// TwinCAT 3 PLC project TcUnitVerifier
// Title: TcUnit verifier
// Company: www.tcunit.org
// Author: Jakob Sagatowski and other contributors, see CONTRIBUTORS file on www.github.com/tcunit/TcUnit-Verifier
// ProjectVersion: 0.5.0.0
// Description: This project is can be used to verify the different functions of TcUnit. It has various test suites to test different functions in TcUnit. By making sure to comment out everything except the test suite that is interesting it is possible to test only the specific function of TcUnit that is interesting.
// ProgramVersion: 3.1.4022.4
// libraries:
//   Tc2_Standard, * (Beckhoff Automation GmbH)
//   Tc2_System, * (Beckhoff Automation GmbH)
//   Tc3_Module, * (Beckhoff Automation GmbH)
//   TcUnit, * (www.tcunit.org)
// project tree:
//   / FB_AdjustAssertFailureMessageToMax252CharLength_Test.TcPOU (not stored), PlcTask.TcTTO
//   Test/ FB_AnyToUnionValue_Test.TcPOU, FB_ArrayPrimitiveTypes_Test.TcPOU, FB_AssertEveryFailedTestTwice.TcPOU, FB_AssertEveryFailedTestTwice_ArrayVersion.TcPOU, FB_CreateFourTestsWithSameName.TcPOU, FB_CreateDisabledTest.TcPOU, FB_MultipleAssertWithSameParametersInDifferentCyclesAndInSameTest.TcPOU, FB_MultipleAssertWithSameParametersInSameCycleWithSameTest.TcPOU, FB_MultipleAssertWithSameParametersInDifferentCyclesButWithDifferentTests.TcPOU, FB_PrimitiveTypes_Test.TcPOU, FB_AssertTrueFalse_Test.TcPOU, FB_AnyPrimitiveTypes_Test.TcPOU, PRG_TEST.TcPOU
// real-time tasks:
//   TASK PlcTask: cycle T#10ms, priority 20, ADS port 350

CONFIGURATION TcUnitVerifier
    RESOURCE PLC ON TwinCAT3
        TASK PlcTask(INTERVAL := T#10ms, PRIORITY := 20);
        PROGRAM PRG_TEST WITH PlcTask : PRG_TEST;
    END_RESOURCE
END_CONFIGURATION

// ---- Test/PRG_TEST.TcPOU
PROGRAM PRG_TEST
VAR
    PrimitiveTypesTest : FB_PrimitiveTypes_Test;
    AssertTrueFalse_Test : FB_AssertTrueFalse_Test;
    AssertEveryFailedTestTwice : FB_AssertEveryFailedTestTwice;
    CreateFourTestsWithSameName : FB_CreateFourTestsWithSameName;
    ArrayPrimitiveTypes_Test : FB_ArrayPrimitiveTypes_Test;
    CreateDisabledTest : FB_CreateDisabledTest;
    AnyPrimitiveTypes_Test : FB_AnyPrimitiveTypes_Test;
    AssertEveryFailedTestTwice_ArrayVersion : FB_AssertEveryFailedTestTwice_ArrayVersion;
    AnyToUnionValue_Test : FB_AnyToUnionValue_Test;
    MultipleAssertWithSameParametersInSameCycleWithSameTest : FB_MultipleAssertWithSameParametersInSameCycleWithSameTest;
    MultipleAssertWithSameParametersInDifferentCyclesButWithDifferentTests : FB_MultipleAssertWithSameParametersInDifferentCyclesButWithDifferentTests;
    MultipleAssertWithSameParametersInDifferentCyclesAndInSameTest : FB_MultipleAssertWithSameParametersInDifferentCyclesAndInSameTest;
END_VAR

TcUnit.RUN();

END_PROGRAM

// ---- Test/FB_PrimitiveTypes_Test.TcPOU
(*
    This testsuite tests the different assert-functions for all the different data types in TwinCAT.
    For every data type at least two different tests have been defined:
        1. One test that succeeds (Expected and actual are equal)
        2. One test that fails (Expected and actual are false).
*)
{attribute 'call_after_init'}
FUNCTION_BLOCK FB_PrimitiveTypes_Test EXTENDS TcUnit.FB_TestSuite

Test_ANY_Equals();
Test_ANY_Differ_DataType();
Test_BYTE_Equals();
Test_BYTE_Differ();
Test_BOOL_Equals();
Test_BOOL_Differ();
Test_DATE_Equals();
Test_DATE_Differ();
Test_DATE_AND_TIME_Equals();
Test_DATE_AND_TIME_Differ();
Test_DINT_Equals();
Test_DINT_Differ();
Test_DWORD_Equals();
Test_DWORD_Differ();
Test_INT_Equals();
Test_INT_Differ();
Test_LINT_Equals();
Test_LINT_Differ();
Test_LREAL_Equals();
Test_LREAL_Differ();
Test_LTIME_Equals();
Test_LTIME_Differ();
Test_LWORD_Equals();
Test_LWORD_Differ();
Test_REAL_Equals();
Test_REAL_Differ();
Test_SINT_Equals();
Test_SINT_Differ();
Test_STRING_Equals();
Test_STRING_Differ();
Test_TIME_Equals();
Test_TIME_Differ();
Test_TIME_OF_DAY_Equals();
Test_TIME_OF_DAY_Differ();
Test_UDINT_Equals();
Test_UDINT_Differ();
Test_UINT_Equals();
Test_UINT_Differ();
Test_ULINT_Equals();
Test_ULINT_Differ();
Test_USINT_Equals();
Test_USINT_Differ();
Test_WORD_Equals();
Test_WORD_Differ();

METHOD PRIVATE Test_ANY_Differ_DataType
VAR
    a : INT := 5;
    b : UINT := 5;
END_VAR
TEST('Test_ANY_Differ_DataType');

AssertEquals(Expected := a,
             Actual := b,
             Message := 'Values differ');

TEST_FINISHED();
END_METHOD

METHOD PRIVATE Test_ANY_Equals
VAR
    a : INT := 5;
    b : INT := 5;
END_VAR
TEST('Test_ANY_Equals');

AssertEquals(Expected := a,
             Actual := b,
             Message := 'Values differ');

TEST_FINISHED();
END_METHOD

METHOD PRIVATE Test_BOOL_Differ
VAR
    a : BOOL := TRUE;
    b : BOOL := FALSE;
END_VAR
TEST('Test_BOOL_Differ');

AssertEquals_BOOL(Expected := a,
                  Actual := b,
                  Message := 'Values differ');

TEST_FINISHED();
END_METHOD

METHOD PRIVATE Test_BOOL_Equals
VAR
    a : BOOL := TRUE;
    b : BOOL := TRUE;
END_VAR
TEST('Test_BOOL_Equals');

AssertEquals_BOOL(Expected := a,
                  Actual := b,
                  Message := 'Values differ');

TEST_FINISHED();
END_METHOD

METHOD PRIVATE Test_BYTE_Differ
VAR
    a : BYTE := 16#AB;
    b : BYTE := 16#CD;
END_VAR
TEST('Test_BYTE_Differ');

AssertEquals_BYTE(Expected := a,
                  Actual := b,
                  Message := 'Values differ');

TEST_FINISHED();
END_METHOD

METHOD PRIVATE Test_BYTE_Equals
VAR
    a : BYTE := 16#CD;
    b : BYTE := 16#CD;
END_VAR
TEST('Test_BYTE_Equals');

AssertEquals_BYTE(Expected := a,
                  Actual := b,
                  Message := 'Values differ');
TEST_FINISHED();
END_METHOD

METHOD PRIVATE Test_DATE_AND_TIME_Differ
VAR
    a : DATE_AND_TIME := DATE_AND_TIME#1996-05-06-15:36:30;
    b : DATE_AND_TIME := DATE_AND_TIME#1972-03-29-00:00:00;
END_VAR
TEST('Test_DATE_AND_TIME_Differ');

AssertEquals_DATE_AND_TIME(Expected := a,
                           Actual := b,
                           Message := 'Values differ');

TEST_FINISHED();
END_METHOD

METHOD PRIVATE Test_DATE_AND_TIME_Equals
VAR
    a : DATE_AND_TIME := DATE_AND_TIME#2019-01-20-13:54:30;
    b : DATE_AND_TIME := DATE_AND_TIME#2019-01-20-13:54:30;
END_VAR
TEST('Test_DATE_AND_TIME_Equals');

AssertEquals_DATE_AND_TIME(Expected := a,
                           Actual := b,
                           Message := 'Values differ');

TEST_FINISHED();
END_METHOD

METHOD PRIVATE Test_DATE_Differ
VAR
    a : DATE := DATE#1996-05-06;
    b : DATE := DATE#2019-01-20;
END_VAR
TEST('Test_DATE_Differ');

AssertEquals_DATE(Expected := a,
                  Actual := b,
                  Message := 'Values differ');

TEST_FINISHED();
END_METHOD

METHOD PRIVATE Test_DATE_Equals
VAR
    a : DATE := DATE#1996-05-06;
    b : DATE := DATE#1996-05-06;
END_VAR
TEST('Test_DATE_Equals');

AssertEquals_DATE(Expected := a,
                  Actual := b,
                  Message := 'Values differ');

TEST_FINISHED();
END_METHOD

METHOD PRIVATE Test_DINT_Differ
VAR
    a : DINT := -55555;
    b : DINT := 70000;
END_VAR
TEST('Test_DINT_Differ');

AssertEquals_DINT(Expected := a,
                  Actual := b,
                  Message := 'Values differ');

TEST_FINISHED();
END_METHOD

METHOD PRIVATE Test_DINT_Equals
VAR
    a : DINT := -80000;
    b : DINT := -80000;
END_VAR
TEST('Test_DINT_Equals');

AssertEquals_DINT(Expected := a,
                  Actual := b,
                  Message := 'Values differ');

TEST_FINISHED();
END_METHOD

METHOD PRIVATE Test_DWORD_Differ
VAR
    a : DWORD := 16#12345678;
    b : DWORD := 16#90ABCDEF;
END_VAR
TEST('Test_DWORD_Differ');

AssertEquals_DWORD(Expected := a,
                   Actual := b,
                   Message := 'Values differ');

TEST_FINISHED();
END_METHOD

METHOD PRIVATE Test_DWORD_Equals
VAR
    a : DWORD := 16#7890ABCD;
    b : DWORD := 16#7890ABCD;
END_VAR
TEST('Test_DWORD_Equals');

AssertEquals_DWORD(Expected := a,
                   Actual := b,
                   Message := 'Values differ');

TEST_FINISHED();
END_METHOD

METHOD PRIVATE Test_INT_Differ
VAR
    a : INT := -32000;
    b : INT := 15423;
END_VAR
TEST('Test_INT_Differ');

AssertEquals_INT(Expected := a,
                 Actual := b,
                 Message := 'Values differ');

TEST_FINISHED();
END_METHOD

METHOD PRIVATE Test_INT_Equals
VAR
    a : INT := -12345;
    b : INT := -12345;
END_VAR
TEST('Test_INT_Equals');

AssertEquals_INT(Expected := a,
                 Actual := b,
                 Message := 'Values differ');

TEST_FINISHED();
END_METHOD

METHOD PRIVATE Test_LINT_Differ
VAR
    a : LINT := -451416345;
    b : LINT := 589532453;
END_VAR
TEST('Test_LINT_Differ');

AssertEquals_LINT(Expected := a,
                  Actual := b,
                  Message := 'Values differ');

TEST_FINISHED();
END_METHOD

METHOD PRIVATE Test_LINT_Equals
VAR
    a : LINT := -123456789;
    b : LINT := -123456789;
END_VAR
TEST('Test_LINT_Equals');

AssertEquals_LINT(Expected := a,
                  Actual := b,
                  Message := 'Values differ');

TEST_FINISHED();
END_METHOD

METHOD PRIVATE Test_LREAL_Differ
VAR
    a : LREAL := 1234567.89;
    b : LREAL := 1234567.76;
END_VAR
TEST('Test_LREAL_Differ');

AssertEquals_LREAL(Expected := a,
                   Actual := b,
                   Delta := 0.1,
                   Message := 'Values differ');

TEST_FINISHED();
END_METHOD

METHOD PRIVATE Test_LREAL_Equals
VAR
    a : LREAL := 1234567.89;
    b : LREAL := 1234567.76;
END_VAR
TEST('Test_LREAL_Equals');

AssertEquals_LREAL(Expected := a,
                   Actual := b,
                   Delta := 0.2,
                   Message := 'Values differ');

TEST_FINISHED();
END_METHOD

METHOD PRIVATE Test_LTIME_Differ
VAR
    a : LTIME := LTIME#213503D23H34M33S709MS551US615NS;
    b : LTIME := LTIME#1000D15H23M12S34MS2US44NS;
END_VAR
TEST('Test_LTIME_Differ');

AssertEquals_LTIME(Expected := a,
                   Actual := b,
                   Message := 'Values differ');

TEST_FINISHED();
END_METHOD

METHOD PRIVATE Test_LTIME_Equals
VAR
    a : LTIME := LTIME#213503D23H34M33S709MS551US615NS;
    b : LTIME := LTIME#213503D23H34M33S709MS551US615NS;
END_VAR
TEST('Test_LTIME_Equals');

AssertEquals_LTIME(Expected := a,
                   Actual := b,
                   Message := 'Values differ');

TEST_FINISHED();
END_METHOD

METHOD PRIVATE Test_LWORD_Differ
VAR
    a : LWORD := 16#0123656789ABCBEC;
    b : LWORD := 16#0123256789ABCAEE;
END_VAR
TEST('Test_LWORD_Differ');

AssertEquals_LWORD(Expected := a,
                   Actual := b,
                   Message := 'Values differ');

TEST_FINISHED();
END_METHOD

METHOD PRIVATE Test_LWORD_Equals
VAR
    a : LWORD := 16#0123456789ABCDEF;
    b : LWORD := 16#0123456789ABCDEF;
END_VAR
TEST('Test_LWORD_Equals');

AssertEquals_LWORD(Expected := a,
                   Actual := b,
                   Message := 'Values differ');

TEST_FINISHED();
END_METHOD

METHOD PRIVATE Test_REAL_Differ
VAR
    a : REAL := 1234.5;
    b : REAL := 1234.4;
END_VAR
TEST('Test_REAL_Differ');

AssertEquals_REAL(Expected := a,
                  Actual := b,
                  Delta := 0.05,
                  Message := 'Values differ');

TEST_FINISHED();
END_METHOD

METHOD PRIVATE Test_REAL_Equals
VAR
    a : REAL := 1234.5;
    b : REAL := 1234.4;
END_VAR
TEST('Test_REAL_Equals');

AssertEquals_REAL(Expected := a,
                  Actual := b,
                  Delta := 0.1,
                  Message := 'Values differ');

TEST_FINISHED();
END_METHOD

METHOD PRIVATE Test_SINT_Differ
VAR
    a : SINT := 127;
    b : SINT := -30;
END_VAR
TEST('Test_SINT_Differ');

AssertEquals_SINT(Expected := a,
                  Actual := b,
                  Message := 'Values differ');

TEST_FINISHED();
END_METHOD

METHOD PRIVATE Test_SINT_Equals
VAR
    a : SINT := -128;
    b : SINT := -128;
END_VAR
TEST('Test_SINT_Equals');

AssertEquals_SINT(Expected := a,
                  Actual := b,
                  Message := 'Values differ');

TEST_FINISHED();
END_METHOD

METHOD PRIVATE Test_STRING_Differ
VAR
    a : STRING := 'This is a string';
    b : STRING := 'This is another string';
END_VAR
TEST('Test_STRING_Differ');

AssertEquals_STRING(Expected := a,
                    Actual := b,
                    Message := 'Values differ');

TEST_FINISHED();
END_METHOD

METHOD PRIVATE Test_STRING_Equals
VAR
    a : STRING := 'Hello there';
    b : STRING := 'Hello there';
END_VAR
TEST('Test_STRING_Equals');

AssertEquals_STRING(Expected := a,
                    Actual := b,
                    Message := 'Values differ');

TEST_FINISHED();
END_METHOD

METHOD PRIVATE Test_TIME_Differ
VAR
    a : TIME := T#12H34M15S10MS;
    b : TIME := T#11H34M13S244MS;
END_VAR
TEST('Test_TIME_Differ');

AssertEquals_TIME(Expected := a,
                  Actual := b,
                  Message := 'Values differ');

TEST_FINISHED();
END_METHOD

METHOD PRIVATE Test_TIME_Equals
VAR
    a : TIME := T#11H34M13S244MS;
    b : TIME := T#11H34M13S244MS;
END_VAR
TEST('Test_TIME_Equals');

AssertEquals_TIME(Expected := a,
                  Actual := b,
                  Message := 'Values differ');

TEST_FINISHED();
END_METHOD

METHOD PRIVATE Test_TIME_OF_DAY_Differ
VAR
    a : TIME_OF_DAY := TIME_OF_DAY#15:36:30.123;
    b : TIME_OF_DAY := TIME_OF_DAY#06:21:11.492;
END_VAR
TEST('Test_TIME_OF_DAY_Differ');

AssertEquals_TIME_OF_DAY(Expected := a,
                         Actual := b,
                         Message := 'Values differ');

TEST_FINISHED();
END_METHOD

METHOD PRIVATE Test_TIME_OF_DAY_Equals
VAR
    a : TIME_OF_DAY := TIME_OF_DAY#06:21:11.492;
    b : TIME_OF_DAY := TIME_OF_DAY#06:21:11.492;
END_VAR
TEST('Test_TIME_OF_DAY_Equals');

AssertEquals_TIME_OF_DAY(Expected := a,
                         Actual := b,
                         Message := 'Values differ');

TEST_FINISHED();
END_METHOD

METHOD PRIVATE Test_UDINT_Differ
VAR
    a : UDINT := 34124214;
    b : UDINT := 52343244;
END_VAR
TEST('Test_UDINT_Differ');

AssertEquals_UDINT(Expected := a,
                   Actual := b,
                   Message := 'Values differ');

TEST_FINISHED();
END_METHOD

METHOD PRIVATE Test_UDINT_Equals
VAR
    a : UDINT := 21845123;
    b : UDINT := 21845123;
END_VAR
TEST('Test_UDINT_Equals');

AssertEquals_UDINT(Expected := a,
                   Actual := b,
                   Message := 'Values differ');

TEST_FINISHED();
END_METHOD

METHOD PRIVATE Test_UINT_Differ
VAR
    a : UINT := 64322;
    b : UINT := 32312;
END_VAR
TEST('Test_UINT_Differ');

AssertEquals_UINT(Expected := a,
                  Actual := b,
                  Message := 'Values differ');

TEST_FINISHED();
END_METHOD

METHOD PRIVATE Test_UINT_Equals
VAR
    a : UINT := 65535;
    b : UINT := 65535;
END_VAR
TEST('Test_UINT_Equals');

AssertEquals_UINT(Expected := a,
                  Actual := b,
                  Message := 'Values differ');

TEST_FINISHED();
END_METHOD

METHOD PRIVATE Test_ULINT_Differ
VAR
    a : ULINT := 10000;
    b : ULINT := 53685437234;
END_VAR
TEST('Test_ULINT_Differ');

AssertEquals_ULINT(Expected := a,
                   Actual := b,
                   Message := 'Values differ');

TEST_FINISHED();
END_METHOD

METHOD PRIVATE Test_ULINT_Equals
VAR
    a : ULINT := 45683838383;
    b : ULINT := 45683838383;
END_VAR
TEST('Test_ULINT_Equals');

AssertEquals_ULINT(Expected := a,
                   Actual := b,
                   Message := 'Values differ');

TEST_FINISHED();
END_METHOD

METHOD PRIVATE Test_USINT_Differ
VAR
    a : USINT := 3;
    b : USINT := 7;
END_VAR
TEST('Test_USINT_Differ');

AssertEquals_USINT(Expected := a,
                   Actual := b,
                   Message := 'Values differ');

TEST_FINISHED();
END_METHOD

METHOD PRIVATE Test_USINT_Equals
VAR
    a : USINT := 5;
    b : USINT := 5;
END_VAR
TEST('Test_USINT_Equals');

AssertEquals_USINT(Expected := a,
                   Actual := b,
                   Message := 'Values differ');

TEST_FINISHED();
END_METHOD

METHOD PRIVATE Test_WORD_Differ
VAR
    a : WORD := 16#EF01;
    b : WORD := 16#2345;
END_VAR
TEST('Test_WORD_Differ');

AssertEquals_WORD(Expected := a,
                  Actual := b,
                  Message := 'Values differ');

TEST_FINISHED();
END_METHOD

METHOD PRIVATE Test_WORD_Equals
VAR
    a : WORD := 16#ABCD;
    b : WORD := 16#ABCD;
END_VAR
TEST('Test_WORD_Equals');

AssertEquals_WORD(Expected := a,
                  Actual := b,
                  Message := 'Values differ');

TEST_FINISHED();
END_METHOD

END_FUNCTION_BLOCK

// ---- Test/FB_AssertTrueFalse_Test.TcPOU
(* 
    This testsuite verifies that the Assert_True and Assert_False methods do what they are supposed to. It does so
    by making sure that every assert-method (assert_true & assert_false) does both one failing and one successful
    assert.
*)
{attribute 'call_after_init'}
FUNCTION_BLOCK FB_AssertTrueFalse_Test EXTENDS TcUnit.FB_TestSuite IMPLEMENTS TcUnit.I_RunnableTestSuite
VAR
    Assert : TcUnit.FB_Assert;
END_VAR

METHOD PRIVATE AssertThatINTsAreEqual
VAR
    a : INT := -33;
    b : INT := -44;
END_VAR
TEST('AssertThatINTsAreEqual');

Assert.AssertFalse(Condition := (a <> b),
                   Message := 'INTs are equal');
END_METHOD

METHOD PRIVATE AssertThatINTsAreNotEqual
VAR
    a : INT := -33;
    b : INT := -44;
END_VAR
TEST('AssertThatINTsAreNotEqual');

Assert.AssertFalse(Condition := (a = b),
                   Message := 'INTs are equal');
END_METHOD

METHOD PRIVATE AssertThatWORDsAreEqual
VAR
    a : WORD := 16#ABCD;
    b : WORD := 16#0123;
END_VAR
TEST('AssertThatWORDsAreEqual');

Assert.AssertTrue(Condition := (a = b),
                  Message := 'WORDs are not equal');
END_METHOD

METHOD PRIVATE AssertThatWORDsAreNotEqual
VAR
    a : WORD := 16#ABCD;
    b : WORD := 16#0123;
END_VAR
TEST('AssertThatWORDsAreNotEqual');

Assert.AssertTrue(Condition := (a <> b),
                  Message := 'WORDs are equal');
END_METHOD

METHOD FB_init : BOOL
VAR_INPUT
	bInitRetains : BOOL; // if TRUE, the retain variables are initialized (warm start / cold start)
	bInCopyCode : BOOL;  // if TRUE, the instance afterwards gets moved into the copy code (online change)
END_VAR
SUPER^.RegisterTestSuite(THIS^);
END_METHOD

METHOD RunTests : TCUNIT.E_TestSuiteRunState
AssertThatINTsAreEqual();
AssertThatINTsAreNotEqual();
AssertThatWORDsAreEqual();
AssertThatWORDsAreNotEqual();

RunTests := TCUNIT.E_TestSuiteRunState.FINISHED;
END_METHOD

END_FUNCTION_BLOCK

// ---- Test/FB_AssertEveryFailedTestTwice.TcPOU
(*
    In this testsuite we are running the same testcase over two cycles, and thus calling every assert method twice.
    This is in order to verify that we don't print every FAILED assert twice.
*)
{attribute 'call_after_init'}
FUNCTION_BLOCK FB_AssertEveryFailedTestTwice EXTENDS TcUnit.FB_TestSuite
VAR
    AssertCount : USINT := 0;
END_VAR

TwiceAssertCall();

METHOD PRIVATE TwiceAssertCall
VAR
    aANY : INT := 55;
    bANY : INT := 77;

    aBOOL : BOOL := TRUE;
    bBOOL : BOOL := FALSE;

    aBYTE : BYTE := 16#AB;
    bBYTE : BYTE := 16#BA;

    aDATE : DATE := DATE#1996-05-06;
    bDATE : DATE := DATE#2019-01-20;

    aDATE_AND_TIME : DATE_AND_TIME := DATE_AND_TIME#1996-05-06-15:36:30;
    bDATE_AND_TIME : DATE_AND_TIME := DATE_AND_TIME#1972-03-29-00:00:00;

    aDINT : DINT := 4444;
    bDINT : DINT := 3333;

    aDWORD : DWORD := 16#AAAAAAAA;
    bDWORD : DWORD := 16#BBBBBBBB;

    aINT : INT := 30000;
    bINT : INT := 32000;

    aLINT : LINT := 50000;
    bLINT : LINT := 50001;

    aLREAL : LREAL := 33.3;
    bLREAL : LREAL := 44.4;

    aLTIME : LTIME := LTIME#213503D23H34M33S709MS551US615NS;
    bLTIME : LTIME := LTIME#1000D15H23M12S34MS2US44NS;

    aLWORD : LWORD := 16#AAAAAAAAAAAAAAAA;
    bLWORD : LWORD := 16#BBBBBBBBBBBBBBBB;

    aREAL : REAL := 44.4;
    bREAL : REAL := 22.2;

    aSINT : SINT := 99;
    bSINT : SINT := 10;

    aSTRING : STRING := 'Hello world';
    bSTRING : STRING := 'Hey there';

    aUDINT : UDINT := 249494994;
    bUDINT : UDINT := 1223;

    aUINT : UINT := 3444;
    bUINT : UINT := 3445;

    aULINT : ULINT := 789234475;
    bULINT : ULINT := 34523327234;

    aUSINT : USINT := 34;
    bUSINT : USINT := 36;

    aTIME : TIME := T#12H34M15S10MS;
    bTIME : TIME := T#11H34M13S244MS;

    aTIME_OF_DAY : TIME_OF_DAY := TIME_OF_DAY#15:36:30.123;
    bTIME_OF_DAY : TIME_OF_DAY := TIME_OF_DAY#06:21:11.492;

    aWORD : WORD := 16#ABCD;
    bWORD : WORD := 16#89EF;
END_VAR
TEST('TwiceAssertCall');

AssertEquals(Expected := aANY,
             Actual := bANY,
             Message := 'Not equal ANY');

AssertEquals_BOOL(Expected := aBOOL,
                  Actual := bBOOL,
                  Message := 'Not equal BOOL');

AssertEquals_BYTE(Expected := aBYTE,
                  Actual := bBYTE,
                  Message := 'Not equal BYTE');

AssertEquals_DATE(Expected := aDATE,
                  Actual := bDATE,
                  Message := 'Not equal DATE');

AssertEquals_DATE_AND_TIME(Expected := aDATE_AND_TIME,
                           Actual := bDATE_AND_TIME,
                           Message := 'Not equal DATE_AND_TIME');

AssertEquals_DINT(Expected := aDINT,
                  Actual := bDINT,
                  Message := 'Not equal DINT');

AssertEquals_DWORD(Expected := aDWORD,
                   Actual := bDWORD,
                   Message := 'Not equal DWORD');

AssertEquals_INT(Expected := aINT,
                 Actual := bINT,
                 Message := 'Not equal INT');

AssertEquals_LINT(Expected := aLINT,
                  Actual := bLINT,
                  Message := 'Not equal LINT');

AssertEquals_LREAL(Expected := aLREAL,
                   Actual := bLREAL,
                   Delta := 0.1,
                   Message := 'Not equal LREAL');

AssertEquals_LTIME(Expected := aLTIME,
                   Actual := bLTIME,
                   Message := 'Not equal LTIME');

AssertEquals_LWORD(Expected := aLWORD,
                   Actual := bLWORD,
                   Message := 'Not equal LWORD');

AssertEquals_REAL(Expected := aREAL,
                  Actual := bREAL,
                  Delta := 0.1,
                  Message := 'Not equal REAL');

AssertEquals_SINT(Expected := aSINT,
                  Actual := bSINT,
                  Message := 'Not equal SINT');

AssertEquals_STRING(Expected := aSTRING,
                    Actual := bSTRING,
                    Message := 'Not equal STRING');

AssertEquals_UDINT(Expected := aUDINT,
                   Actual := bUDINT,
                   Message := 'Not equal UDINT');

AssertEquals_UINT(Expected := aUINT,
                  Actual := bUINT,
                  Message := 'Not equal UINT');

AssertEquals_ULINT(Expected := aULINT,
                   Actual := bULINT,
                   Message := 'Not equal ULINT');

AssertEquals_USINT(Expected := aUSINT,
                   Actual := bUSINT,
                   Message := 'Not equal USINT');

AssertEquals_TIME(Expected := aTIME,
                  Actual := bTIME,
                  Message := 'Not equal TIME');

AssertEquals_TIME_OF_DAY(Expected := aTIME_OF_DAY,
                         Actual := bTIME_OF_DAY,
                         Message := 'Not equal TIME_OF_DAY');

AssertEquals_WORD(Expected := aWORD,
                  Actual := bWORD,
                  Message := 'Not equal WORD');

AssertCount := AssertCount + 1;
IF AssertCount = 2 THEN
    TEST_FINISHED();
END_IF
END_METHOD

END_FUNCTION_BLOCK

// ---- Test/FB_CreateFourTestsWithSameName.TcPOU
(*
    This testsuite creates four tests in the same testsuite with the same name. Every test in a testsuite should have
    an unique name. Every assert should be ignored if a duplicate test is being run.
*)
{attribute 'call_after_init'}
FUNCTION_BLOCK FB_CreateFourTestsWithSameName EXTENDS TcUnit.FB_TestSuite

TestOne();
TestOne_Again();
TestOne_AgainAgain();
TestOne_AgainAgainAgain();

METHOD PRIVATE TestOne
VAR
    a : INT := 55;
    b : INT := 55;
END_VAR
TEST('TestOne');

AssertEquals_INT(Expected := a,
                 Actual := b,
                 Message := 'A does not equal B');

TEST_FINISHED();
END_METHOD

METHOD PRIVATE TestOne_Again
VAR
    a : INT := 55;
    b : INT := 54;
END_VAR
TEST('TestOne');

AssertEquals_INT(Expected := a,
                 Actual := b,
                 Message := 'A does not equal B again');

TEST_FINISHED();
END_METHOD

METHOD PRIVATE TestOne_AgainAgain
VAR
    a : INT := 55;
    b : INT := 55;
END_VAR
TEST('TestOne');

AssertEquals_INT(Expected := a,
                 Actual := b,
                 Message := 'A does not equal B again');

TEST_FINISHED();
END_METHOD

METHOD PRIVATE TestOne_AgainAgainAgain
VAR
    a : INT := 55;
    b : INT := 55;
END_VAR
TEST('TestOne');

AssertEquals_INT(Expected := a,
                 Actual := b,
                 Message := 'A does not equal B again');

TEST_FINISHED();
END_METHOD

END_FUNCTION_BLOCK

// ---- Test/FB_ArrayPrimitiveTypes_Test.TcPOU
(*
    This testsuite tests the different assert-functions for all the different type of arrays (varying by the different
    data types that are available in TwinCAT). For every type of array (BOOL, BYTE, INT etc.) at least three different
    tests have been defined:
        1. One test that succeeds, where the data and size of the arrays are matching
        2. One test that fails, where the size of the arrays differs
        3. One test that fails, where the content of the array differs
*)
{attribute 'call_after_init'}
FUNCTION_BLOCK FB_ArrayPrimitiveTypes_Test EXTENDS TcUnit.FB_TestSuite IMPLEMENTS TcUnit.I_RunnableTestSuite
VAR
    Assert : TcUnit.FB_Assert;
END_VAR

METHOD FB_init : BOOL
VAR_INPUT
	bInitRetains : BOOL; // if TRUE, the retain variables are initialized (warm start / cold start)
	bInCopyCode : BOOL;  // if TRUE, the instance afterwards gets moved into the copy code (online change)
END_VAR
SUPER^.RegisterTestSuite(THIS^);
END_METHOD

METHOD RunTests : TCUNIT.E_TestSuiteRunState
Test_BOOL_Array_Equals();
Test_BOOL_Array_DiffersInSize();
Test_BOOL_Array_DiffersInContent();
Test_BYTE_Array_Equals();
Test_BYTE_Array_DiffersInSize();
Test_BYTE_Array_DiffersInContent();
Test_DINT_Array_Equals();
Test_DINT_Array_DifferInSize();
Test_DINT_Array_DifferInContent();
Test_DWORD_Array_Equals();
Test_DWORD_Array_DifferInSize();
Test_DWORD_Array_DifferInContent();
Test_INT_Array_Equals();
Test_INT_Array_DifferInSize();
Test_INT_Array_DifferInContent();
Test_LINT_Array_Equals();
Test_LINT_Array_DifferInSize();
Test_LINT_Array_DifferInContent();
Test_LWORD_Array_Equals();
Test_LWORD_Array_DifferInSize();
Test_LWORD_Array_DifferInContent();
Test_SINT_Array_Equals();
Test_SINT_Array_DifferInSize();
Test_SINT_Array_DifferInContent();
Test_UDINT_Array_Equals();
Test_UDINT_Array_DifferInSize();
Test_UDINT_Array_DifferInContent();
Test_UINT_Array_Equals();
Test_UINT_Array_DifferInSize();
Test_UINT_Array_DifferInContent();
Test_ULINT_Array_Equals();
Test_ULINT_Array_DifferInSize();
Test_ULINT_Array_DifferInContent();
Test_USINT_Array_Equals();
Test_USINT_Array_DifferInSize();
Test_USINT_Array_DifferInContent();
Test_WORD_Array_Equals();
Test_WORD_Array_DifferInSize();
Test_WORD_Array_DifferInContent();

RunTests := TCUNIT.E_TestSuiteRunState.FINISHED;
END_METHOD

METHOD PRIVATE Test_BOOL_Array_DiffersInContent
VAR
    a : ARRAY[0..5] OF BOOL := [TRUE, TRUE, FALSE, TRUE, FALSE, TRUE];
    b : ARRAY[0..5] OF BOOL := [TRUE, TRUE, TRUE, TRUE, FALSE, FALSE];
END_VAR
TEST('Test_BOOL_Array_DiffersInContent');

Assert.AssertArrayEquals_BOOL(Expecteds := a,
                              Actuals := b,
                              Message := 'Arrays differ');
END_METHOD

METHOD PRIVATE Test_BOOL_Array_DiffersInSize
VAR
    a : ARRAY[1..6] OF BOOL := [TRUE, TRUE, TRUE, TRUE, TRUE, TRUE];
    b : ARRAY[1..4] OF BOOL := [TRUE, TRUE, TRUE, TRUE];
END_VAR
TEST('Test_BOOL_Array_DiffersInSize');

Assert.AssertArrayEquals_BOOL(Expecteds := a,
                              Actuals := b,
                              Message := 'Arrays differ');
END_METHOD

METHOD PRIVATE Test_BOOL_Array_Equals
VAR
    a : ARRAY[1..5] OF BOOL := [TRUE, FALSE, TRUE, FALSE, TRUE];
    b : ARRAY[1..5] OF BOOL := [TRUE, FALSE, TRUE, FALSE, TRUE];
END_VAR
TEST('Test_BOOL_Array_Equals');

Assert.AssertArrayEquals_BOOL(Expecteds := a,
                              Actuals := b,
                              Message := 'Arrays differ');
END_METHOD

METHOD PRIVATE Test_BYTE_Array_DiffersInContent
VAR
    a : ARRAY[0..3] OF BYTE := [16#AB, 16#AA, 16#BB, 16#89];
    b : ARRAY[0..3] OF BYTE := [16#AB, 16#CD, 16#BB, 16#89];
END_VAR
TEST('Test_BYTE_Array_DiffersInContent');

Assert.AssertArrayEquals_BYTE(Expecteds := a,
                              Actuals := b,
                              Message := 'Arrays differ');
END_METHOD

METHOD PRIVATE Test_BYTE_Array_DiffersInSize
VAR
    a : ARRAY[1..2] OF BYTE := [16#AB, 16#CD];
    b : ARRAY[1..5] OF BYTE := [16#AB, 16#CD, 16#EF, 16#01, 16#23];
END_VAR
TEST('Test_BYTE_Array_DiffersInSize');

Assert.AssertArrayEquals_BYTE(Expecteds := a,
                              Actuals := b,
                              Message := 'Arrays differ');
END_METHOD

METHOD PRIVATE Test_BYTE_Array_Equals
VAR
    a : ARRAY[1..3] OF BYTE := [16#FD, 16#34, 16#9E];
    b : ARRAY[1..3] OF BYTE := [16#FD, 16#34, 16#9E];
END_VAR
TEST('Test_BYTE_Array_Equals');

Assert.AssertArrayEquals_BYTE(Expecteds := a,
                              Actuals := b,
                              Message := 'Arrays differ');
END_METHOD

METHOD PRIVATE Test_DINT_Array_DifferInContent
VAR
    a : ARRAY[3..5] OF DINT := [-4746, -2147483645, 0];
    b : ARRAY[3..5] OF DINT := [-4746, -2147483641, 0];
END_VAR
TEST('Test_DINT_Array_DifferInContent');

Assert.AssertArrayEquals_DINT(Expecteds := a,
                              Actuals := b,
                              Message := 'Arrays differ');
END_METHOD

METHOD PRIVATE Test_DINT_Array_DifferInSize
VAR
    a : ARRAY[3..4] OF DINT := [-11, 2147483647];
    b : ARRAY[4..6] OF DINT := [-11, 2147483647, 0];
END_VAR
TEST('Test_DINT_Array_DifferInSize');

Assert.AssertArrayEquals_DINT(Expecteds := a,
                              Actuals := b,
                              Message := 'Arrays differ');
END_METHOD

METHOD PRIVATE Test_DINT_Array_Equals
VAR
    a : ARRAY[2..7] OF DINT := [64, 98, 2147483647, -2147483648, 0, -63987538];
    b : ARRAY[2..7] OF DINT := [64, 98, 2147483647, -2147483648, 0, -63987538];
END_VAR
TEST('Test_DINT_Array_Equals');

Assert.AssertArrayEquals_DINT(Expecteds := a,
                              Actuals := b,
                              Message := 'Arrays differ');
END_METHOD

METHOD PRIVATE Test_DWORD_Array_DifferInContent
VAR
    a : ARRAY[-2..1] OF DWORD := [16#6789ABCD, 16#EFAA2346, 16#ABABABAB, 16#EEEEEEEE];
    b : ARRAY[-2..1] OF DWORD := [16#6789ABCD, 16#EF012345, 16#ABABABAB, 16#EEEEEEEE];
END_VAR
TEST('Test_DWORD_Array_DifferInContent');

Assert.AssertArrayEquals_DWORD(Expecteds := a,
                               Actuals := b,
                               Message := 'Arrays differ');
END_METHOD

METHOD PRIVATE Test_DWORD_Array_DifferInSize
VAR
    a : ARRAY[-2..1] OF DWORD := [16#6789ABCD, 16#EF012345, 16#67890ABC, 16#DDDDDDDD];
    b : ARRAY[-3..-2] OF DWORD := [16#6789ABCD, 16#EF012345];
END_VAR
TEST('Test_DWORD_Array_DifferInSize');

Assert.AssertArrayEquals_DWORD(Expecteds := a,
                               Actuals := b,
                               Message := 'Arrays differ');
END_METHOD

METHOD PRIVATE Test_DWORD_Array_Equals
VAR
    a : ARRAY[2..3] OF DWORD := [16#6789ABCD, 16#EF012345];
    b : ARRAY[1..2] OF DWORD := [16#6789ABCD, 16#EF012345];
END_VAR
TEST('Test_DWORD_Array_Equals');

Assert.AssertArrayEquals_DWORD(Expecteds := a,
                               Actuals := b,
                               Message := 'Arrays differ');
END_METHOD

METHOD PRIVATE Test_INT_Array_DifferInContent
VAR
    a : ARRAY[-8..-6] OF INT := [42, -23, -32768];
    b : ARRAY[1..3] OF INT := [42, 24, -32768];
END_VAR
TEST('Test_INT_Array_DifferInContent');

Assert.AssertArrayEquals_INT(Expecteds := a,
                             Actuals := b,
                             Message := 'Arrays differ');
END_METHOD

METHOD PRIVATE Test_INT_Array_DifferInSize
VAR
    a : ARRAY[-4..3] OF INT := [64, 98, -32768, 32767, 5478, -378, 42, 6234];
    b : ARRAY[1..5] OF INT := [64, 98, -32768, 32767, 5478];
END_VAR
TEST('Test_INT_Array_DifferInSize');

Assert.AssertArrayEquals_INT(Expecteds := a,
                             Actuals := b,
                             Message := 'Arrays differ');
END_METHOD

METHOD PRIVATE Test_INT_Array_Equals
VAR
    a : ARRAY[-5..1] OF INT := [64, 98, -32768, 32767, 5478, -378, 42];
    b : ARRAY[1..7] OF INT := [64, 98, -32768, 32767, 5478, -378, 42];
END_VAR
TEST('Test_INT_Array_Equals');

Assert.AssertArrayEquals_INT(Expecteds := a,
                             Actuals := b,
                             Message := 'Arrays differ');
END_METHOD

METHOD PRIVATE Test_LINT_Array_DifferInContent
VAR
    a : ARRAY[-1..1] OF LINT := [9_223_372_036_854_775_807, -9_223_372_036_853_775_808, 55];
    b : ARRAY[4..6] OF LINT := [9_223_372_036_854_775_807, -9_223_372_036_854_775_808, 55];
END_VAR
TEST('Test_LINT_Array_DifferInContent');

Assert.AssertArrayEquals_LINT(Expecteds := a,
                              Actuals := b,
                              Message := 'Arrays differ');
END_METHOD

METHOD PRIVATE Test_LINT_Array_DifferInSize
VAR
    a : ARRAY[-1..1] OF LINT := [9_223_372_036_854_775_807, -9_223_372_036_854_775_808, 55];
    b : ARRAY[4..5] OF LINT := [9_223_372_036_854_775_807, -9_223_372_036_854_775_808];
END_VAR
TEST('Test_LINT_Array_DifferInSize');

Assert.AssertArrayEquals_LINT(Expecteds := a,
                              Actuals := b,
                              Message := 'Arrays differ');
END_METHOD

METHOD PRIVATE Test_LINT_Array_Equals
VAR
    a : ARRAY[-1..0] OF LINT := [9_223_372_036_854_775_807, -9_223_372_036_854_775_808];
    b : ARRAY[4..5] OF LINT := [9_223_372_036_854_775_807, -9_223_372_036_854_775_808];
END_VAR
TEST('Test_LINT_Array_Equals');

Assert.AssertArrayEquals_LINT(Expecteds := a,
                              Actuals := b,
                              Message := 'Arrays differ');
END_METHOD

METHOD PRIVATE Test_LWORD_Array_DifferInContent
VAR
    a : ARRAY[1..1] OF LWORD := [16#EDCBA09876543210];
    b : ARRAY[1..1] OF LWORD := [16#01234567890ABCDE];
END_VAR
TEST('Test_LWORD_Array_DifferInContent');

Assert.AssertArrayEquals_LWORD(Expecteds := a,
                               Actuals := b,
                               Message := 'Arrays differ');
END_METHOD

METHOD PRIVATE Test_LWORD_Array_DifferInSize
VAR
    a : ARRAY[1..1] OF LWORD := [16#EDCBA09876543210];
    b : ARRAY[1..2] OF LWORD := [16#01234567890ABCDE, 16#EDCBA09876543210];
END_VAR
TEST('Test_LWORD_Array_DifferInSize');

Assert.AssertArrayEquals_LWORD(Expecteds := a,
                               Actuals := b,
                               Message := 'Arrays differ');
END_METHOD

METHOD PRIVATE Test_LWORD_Array_Equals
VAR
    a : ARRAY[1..2] OF LWORD := [16#01234567890ABCDE, 16#EDCBA09876543210];
    b : ARRAY[1..2] OF LWORD := [16#01234567890ABCDE, 16#EDCBA09876543210];
END_VAR
TEST('Test_LWORD_Array_Equals');

Assert.AssertArrayEquals_LWORD(Expecteds := a,
                               Actuals := b,
                               Message := 'Arrays differ');
END_METHOD

METHOD PRIVATE Test_SINT_Array_DifferInContent
VAR
    a : ARRAY[0..0] OF SINT := [-128];
    b : ARRAY[0..0] OF SINT := [127];
END_VAR
TEST('Test_SINT_Array_DifferInContent');

Assert.AssertArrayEquals_SINT(Expecteds := a,
                              Actuals := b,
                              Message := 'Arrays differ');
END_METHOD

METHOD PRIVATE Test_SINT_Array_DifferInSize
VAR
    a : ARRAY[0..0] OF SINT := [-128];
    b : ARRAY[0..1] OF SINT := [-128, 127];
END_VAR
TEST('Test_SINT_Array_DifferInSize');

Assert.AssertArrayEquals_SINT(Expecteds := a,
                              Actuals := b,
                              Message := 'Arrays differ');
END_METHOD

METHOD PRIVATE Test_SINT_Array_Equals
VAR
    a : ARRAY[0..3] OF SINT := [-128, 127, -34, 62];
    b : ARRAY[0..3] OF SINT := [-128, 127, -34, 62];
END_VAR
TEST('Test_SINT_Array_Equals');

Assert.AssertArrayEquals_SINT(Expecteds := a,
                              Actuals := b,
                              Message := 'Arrays differ');
END_METHOD

METHOD PRIVATE Test_UDINT_Array_DifferInContent
VAR
    a : ARRAY[-5..-4] OF UDINT := [4294967295, 5];
    b : ARRAY[0..1] OF UDINT := [4294967295, 4];
END_VAR
TEST('Test_UDINT_Array_DifferInContent');

Assert.AssertArrayEquals_UDINT(Expecteds := a,
                               Actuals := b,
                               Message := 'Arrays differ');
END_METHOD

METHOD PRIVATE Test_UDINT_Array_DifferInSize
VAR
    a : ARRAY[-5..-4] OF UDINT := [4294967295, 0];
    b : ARRAY[0..2] OF UDINT := [4294967295, 0, 5000];
END_VAR
TEST('Test_UDINT_Array_DifferInSize');

Assert.AssertArrayEquals_UDINT(Expecteds := a,
                               Actuals := b,
                               Message := 'Arrays differ');
END_METHOD

METHOD PRIVATE Test_UDINT_Array_Equals
VAR
    a : ARRAY[1..3] OF UDINT := [0, 4294967295, 5000];
    b : ARRAY[1..3] OF UDINT := [0, 4294967295, 5000];
END_VAR
TEST('Test_UDINT_Array_Equals');

Assert.AssertArrayEquals_UDINT(Expecteds := a,
                               Actuals := b,
                               Message := 'Arrays differ');
END_METHOD

METHOD PRIVATE Test_UINT_Array_DifferInContent
VAR
    a : ARRAY[0..3] OF UINT := [0, 4, 8, 99];
    b : ARRAY[0..3] OF UINT := [0, 4, 8, 12];
END_VAR
TEST('Test_UINT_Array_DifferInContent');

Assert.AssertArrayEquals_UINT(Expecteds := a,
                              Actuals := b,
                              Message := 'Arrays differ');
END_METHOD

METHOD PRIVATE Test_UINT_Array_DifferInSize
VAR
    a : ARRAY[0..2] OF UINT := [0, 4, 8];
    b : ARRAY[0..3] OF UINT := [0, 4, 8, 12];
END_VAR
TEST('Test_UINT_Array_DifferInSize');

Assert.AssertArrayEquals_UINT(Expecteds := a,
                              Actuals := b,
                              Message := 'Arrays differ');
END_METHOD

METHOD PRIVATE Test_UINT_Array_Equals
VAR
    a : ARRAY[0..4] OF UINT := [0, 65535, 2000, 34123, 59];
    b : ARRAY[0..4] OF UINT := [0, 65535, 2000, 34123, 59];
END_VAR
TEST('Test_UINT_Array_Equals');

Assert.AssertArrayEquals_UINT(Expecteds := a,
                              Actuals := b,
                              Message := 'Arrays differ');
END_METHOD

METHOD PRIVATE Test_ULINT_Array_DifferInContent
VAR
    a : ARRAY[0..1] OF ULINT := [3_213_000_444_000, 9_400_000_000_000];
    b : ARRAY[0..1] OF ULINT := [3_213_000_444_000, 18_446_744_073_709_551_615];
END_VAR
TEST('Test_ULINT_Array_DifferInContent');

Assert.AssertArrayEquals_ULINT(Expecteds := a,
                               Actuals := b,
                               Message := 'Arrays differ');
END_METHOD

METHOD PRIVATE Test_ULINT_Array_DifferInSize
VAR
    a : ARRAY[0..1] OF ULINT := [0, 9_400_000_000_000];
    b : ARRAY[0..0] OF ULINT := [0];
END_VAR
TEST('Test_ULINT_Array_DifferInSize');

Assert.AssertArrayEquals_ULINT(Expecteds := a,
                               Actuals := b,
                               Message := 'Arrays differ');
END_METHOD

METHOD PRIVATE Test_ULINT_Array_Equals
VAR
    a : ARRAY[0..3] OF ULINT := [0, 18_446_744_073_709_551_615, 9_400_000_000_000, 3_213_000_444_000];
    b : ARRAY[0..3] OF ULINT := [0, 18_446_744_073_709_551_615, 9_400_000_000_000, 3_213_000_444_000];
END_VAR
TEST('Test_ULINT_Array_Equals');

Assert.AssertArrayEquals_ULINT(Expecteds := a,
                               Actuals := b,
                               Message := 'Arrays differ');
END_METHOD

METHOD PRIVATE Test_USINT_Array_DifferInContent
VAR
    a : ARRAY[0..10] OF USINT := [0,1,2,3,6(4),5];
    b : ARRAY[0..10] OF USINT := [0,1,2,3,6(5),6];
END_VAR
TEST('Test_USINT_Array_DifferInContent');

Assert.AssertArrayEquals_USINT(Expecteds := a,
                               Actuals := b,
                               Message := 'Arrays differ');
END_METHOD

METHOD PRIVATE Test_USINT_Array_DifferInSize
VAR
    a : ARRAY[0..100] OF USINT := [101(42)];
    b : ARRAY[0..70] OF USINT := [71(42)];
END_VAR
TEST('Test_USINT_Array_DifferInSize');

Assert.AssertArrayEquals_USINT(Expecteds := a,
                               Actuals := b,
                               Message := 'Arrays differ');
END_METHOD

METHOD PRIVATE Test_USINT_Array_Equals
VAR
    a : ARRAY[0..100] OF USINT := [42, 100(33)];
    b : ARRAY[0..100] OF USINT := [42, 100(33)];
END_VAR
TEST('Test_USINT_Array_Equals');

Assert.AssertArrayEquals_USINT(Expecteds := a,
                               Actuals := b,
                               Message := 'Arrays differ');
END_METHOD

METHOD PRIVATE Test_WORD_Array_DifferInContent
VAR
    a : ARRAY[1..7] OF WORD := [16#2323, 16#876A, 16#4CD4, 16#F3DC, 16#BBBB, 16#FFFF, 16#1133];
    b : ARRAY[1..7] OF WORD := [16#2323, 16#876A, 16#4CD4, 16#F3DC, 16#BBBB, 16#FFFF, 16#1122];
END_VAR
TEST('Test_WORD_Array_DifferInContent');

Assert.AssertArrayEquals_WORD(Expecteds := a,
                              Actuals := b,
                              Message := 'Arrays differ');
END_METHOD

METHOD PRIVATE Test_WORD_Array_DifferInSize
VAR
    a : ARRAY[1..5] OF WORD := [16#0000, 16#3333, 16#5555, 16#7777, 16#BBBB];
    b : ARRAY[1..7] OF WORD := [16#0000, 16#3333, 16#5555, 16#7777, 16#BBBB, 16#FFFF, 16#1122];
END_VAR
TEST('Test_WORD_Array_DifferInSize');

Assert.AssertArrayEquals_WORD(Expecteds := a,
                              Actuals := b,
                              Message := 'Arrays differ');
END_METHOD

METHOD PRIVATE Test_WORD_Array_Equals
VAR
    a : ARRAY[1..5] OF WORD := [16#AAAA, 16#BBBB, 16#CCCC, 16#DDDD, 16#EEEE];
    b : ARRAY[1..5] OF WORD := [16#AAAA, 16#BBBB, 16#CCCC, 16#DDDD, 16#EEEE];
END_VAR
TEST('Test_WORD_Array_Equals');

Assert.AssertArrayEquals_WORD(Expecteds := a,
                              Actuals := b,
                              Message := 'Arrays differ');
END_METHOD

END_FUNCTION_BLOCK

// ---- Test/FB_CreateDisabledTest.TcPOU
(*
    This testsuite runs two tests. One that is enabled (and that is supposed to fail), and one that is disabled (and
    even though it also is failing is not supposed to run).
*)
{attribute 'call_after_init'}
FUNCTION_BLOCK FB_CreateDisabledTest EXTENDS TcUnit.FB_TestSuite

TestEnabled();
TestDisabled();

METHOD PRIVATE TestDisabled
VAR
    a : BOOL := FALSE;
    b : BOOL := TRUE;
END_VAR
TEST('DISABLED_ThisShouldNotExecute');

AssertEquals(Expected := a,
             Actual := b,
             Message := 'A does not equal B');

TEST_FINISHED();
END_METHOD

METHOD PRIVATE TestEnabled
VAR
    a : BOOL := TRUE;
    b : BOOL := FALSE;
END_VAR
TEST('TestEnabled');

AssertEquals(Expected := a,
             Actual := b,
             Message := 'A does not equal B');

TEST_FINISHED();
END_METHOD

END_FUNCTION_BLOCK

// ---- Test/FB_AnyPrimitiveTypes_Test.TcPOU
(*
    This testsuite tests the different assert-functions for all the primitive data types in TwinCAT, but using the
    ANY-version of the Assert-method.
    For every data type at least two different tests have been defined:
        1. One test that succeeds (Expected and actual are equal)
        2. One test that fails (Expected and actual are false).
    For every failing test the printed value should be the same as if we were using the primitive data type assert
    directly. 
*)
{attribute 'call_after_init'}
FUNCTION_BLOCK FB_AnyPrimitiveTypes_Test EXTENDS TcUnit.FB_TestSuite

Test_ANY_BYTE_Equals();
Test_ANY_BYTE_Differ();
Test_ANY_BOOL_Equals();
Test_ANY_BOOL_Differ();
Test_ANY_DATE_Equals();
Test_ANY_DATE_Differ();
Test_ANY_DATE_AND_TIME_Equals();
Test_ANY_DATE_AND_TIME_Differ();
Test_ANY_DINT_Equals();
Test_ANY_DINT_Differ();
Test_ANY_DWORD_Equals();
Test_ANY_DWORD_Differ();
Test_ANY_INT_Equals();
Test_ANY_INT_Differ();
Test_ANY_LINT_Equals();
Test_ANY_LINT_Differ();
Test_ANY_LREAL_Equals();
Test_ANY_LREAL_Differ();
Test_ANY_LTIME_Equals();
Test_ANY_LTIME_Differ();
Test_ANY_LWORD_Equals();
Test_ANY_LWORD_Differ();
Test_ANY_REAL_Equals();
Test_ANY_REAL_Differ();
Test_ANY_SINT_Equals();
Test_ANY_SINT_Differ();
Test_ANY_STRING_Equals();
Test_ANY_STRING_Differ();
Test_ANY_TIME_Equals();
Test_ANY_TIME_Differ();
Test_ANY_TIME_OF_DAY_Equals();
TesT_ANY_TIME_OF_DAY_Differ();
Test_ANY_UDINT_Equals();
Test_ANY_UDINT_Differ();
Test_ANY_UINT_Equals();
Test_ANY_UINT_Differ();
Test_ANY_ULINT_Equals();
Test_ANY_ULINT_Differ();
Test_ANY_USINT_Equals();
Test_ANY_USINT_Differ();
Test_ANY_WORD_Equals();
Test_ANY_WORD_Differ();

METHOD PRIVATE Test_ANY_BOOL_Differ
VAR
    a : BOOL := TRUE;
    b : BOOL := FALSE;
END_VAR
TEST('Test_ANY_BOOL_Differ');

AssertEquals(Expected := a,
             Actual := b,
             Message := 'Values differ');

TEST_FINISHED();
END_METHOD

METHOD PRIVATE Test_ANY_BOOL_Equals
VAR
    a : BOOL := TRUE;
    b : BOOL := TRUE;
END_VAR
TEST('Test_ANY_BOOL_Equals');

AssertEquals(Expected := a,
             Actual := b,
             Message := 'Values differ');

TEST_FINISHED();
END_METHOD

METHOD PRIVATE Test_ANY_BYTE_Differ
VAR
    a : BYTE := 16#AB;
    b : BYTE := 16#CD;
END_VAR
TEST('Test_ANY_BYTE_Differ');

AssertEquals(Expected := a,
             Actual := b,
             Message := 'Values differ');

TEST_FINISHED();
END_METHOD

METHOD PRIVATE Test_ANY_BYTE_Equals
VAR
    a : BYTE := 16#CD;
    b : BYTE := 16#CD;
END_VAR
TEST('Test_ANY_BYTE_Equals');

AssertEquals(Expected := a,
             Actual := b,
             Message := 'Values differ');

TEST_FINISHED();
END_METHOD

METHOD PRIVATE Test_ANY_DATE_AND_TIME_Differ
VAR
    a : DATE_AND_TIME := DATE_AND_TIME#1996-05-06-15:36:30;
    b : DATE_AND_TIME := DATE_AND_TIME#1972-03-29-00:00:00;
END_VAR
TEST('Test_ANY_DATE_AND_TIME_Differ');

AssertEquals(Expected := a,
             Actual := b,
             Message := 'Values differ');

TEST_FINISHED();
END_METHOD

METHOD PRIVATE Test_ANY_DATE_AND_TIME_Equals
VAR
    a : DATE_AND_TIME := DATE_AND_TIME#2019-01-20-13:54:30;
    b : DATE_AND_TIME := DATE_AND_TIME#2019-01-20-13:54:30;
END_VAR
TEST('Test_ANY_DATE_AND_TIME_Equals');

AssertEquals(Expected := a,
             Actual := b,
             Message := 'Values differ');

TEST_FINISHED();
END_METHOD

METHOD PRIVATE Test_ANY_DATE_Differ
VAR
    a : DATE := DATE#1996-05-06;
    b : DATE := DATE#2019-01-20;
END_VAR
TEST('Test_ANY_DATE_Differ');

AssertEquals(Expected := a,
             Actual := b,
             Message := 'Values differ');

TEST_FINISHED();
END_METHOD

METHOD PRIVATE Test_ANY_DATE_Equals
VAR
    a : DATE := DATE#1996-05-06;
    b : DATE := DATE#1996-05-06;
END_VAR
TEST('Test_ANY_DATE_Equals');

AssertEquals(Expected := a,
             Actual := b,
             Message := 'Values differ');

TEST_FINISHED();
END_METHOD

METHOD PRIVATE Test_ANY_DINT_Differ
VAR
    a : DINT := -55555;
    b : DINT := 70000;
END_VAR
TEST('Test_ANY_DINT_Differ');

AssertEquals(Expected := a,
             Actual := b,
             Message := 'Values differ');

TEST_FINISHED();
END_METHOD

METHOD PRIVATE Test_ANY_DINT_Equals
VAR
    a : DINT := -80000;
    b : DINT := -80000;
END_VAR
TEST('Test_ANY_DINT_Equals');

AssertEquals(Expected := a,
             Actual := b,
             Message := 'Values differ');

TEST_FINISHED();
END_METHOD

METHOD PRIVATE Test_ANY_DWORD_Differ
VAR
    a : DWORD := 16#12345678;
    b : DWORD := 16#90ABCDEF;
END_VAR
TEST('Test_ANY_DWORD_Differ');

AssertEquals(Expected := a,
             Actual := b,
             Message := 'Values differ');

TEST_FINISHED();
END_METHOD

METHOD PRIVATE Test_ANY_DWORD_Equals
VAR
    a : DWORD := 16#7890ABCD;
    b : DWORD := 16#7890ABCD;
END_VAR
TEST('Test_ANY_DWORD_Equals');

AssertEquals(Expected := a,
             Actual := b,
             Message := 'Values differ');

TEST_FINISHED();
END_METHOD

METHOD PRIVATE Test_ANY_INT_Differ
VAR
    a : INT := -32000;
    b : INT := 15423;
END_VAR
TEST('Test_ANY_INT_Differ');

AssertEquals(Expected := a,
             Actual := b,
             Message := 'Values differ');

TEST_FINISHED();
END_METHOD

METHOD PRIVATE Test_ANY_INT_Equals
VAR
    a : INT := -12345;
    b : INT := -12345;
END_VAR
TEST('Test_ANY_INT_Equals');

AssertEquals(Expected := a,
             Actual := b,
             Message := 'Values differ');

TEST_FINISHED();
END_METHOD

METHOD PRIVATE Test_ANY_LINT_Differ
VAR
    a : LINT := -451416345;
    b : LINT := 589532453;
END_VAR
TEST('Test_ANY_LINT_Differ');

AssertEquals(Expected := a,
             Actual := b,
             Message := 'Values differ');

TEST_FINISHED();
END_METHOD

METHOD PRIVATE Test_ANY_LINT_Equals
VAR
    a : LINT := -123456789;
    b : LINT := -123456789;
END_VAR
TEST('Test_ANY_LINT_Equals');

AssertEquals(Expected := a,
             Actual := b,
             Message := 'Values differ');

TEST_FINISHED();
END_METHOD

METHOD PRIVATE Test_ANY_LREAL_Differ
VAR
    a : LREAL := 1234567.89;
    b : LREAL := 1234567.76;
END_VAR
TEST('Test_ANY_LREAL_Differ');

AssertEquals(Expected := a,
             Actual := b,
             Message := 'Values differ');

TEST_FINISHED();
END_METHOD

METHOD PRIVATE Test_ANY_LREAL_Equals
VAR
    a : LREAL := 1234567.89;
    b : LREAL := 1234567.89;
END_VAR
TEST('Test_ANY_LREAL_Equals');

AssertEquals(Expected := a,
             Actual := b,
             Message := 'Values differ');

TEST_FINISHED();
END_METHOD

METHOD PRIVATE Test_ANY_LTIME_Differ
VAR
    a : LTIME := LTIME#213503D23H34M33S709MS551US615NS;
    b : LTIME := LTIME#1000D15H23M12S34MS2US44NS;
END_VAR
TEST('Test_ANY_LTIME_Differ');

AssertEquals(Expected := a,
             Actual := b,
             Message := 'Values differ');

TEST_FINISHED();
END_METHOD

METHOD PRIVATE Test_ANY_LTIME_Equals
VAR
    a : LTIME := LTIME#213503D23H34M33S709MS551US615NS;
    b : LTIME := LTIME#213503D23H34M33S709MS551US615NS;
END_VAR
TEST('Test_ANY_LTIME_Equals');

AssertEquals(Expected := a,
             Actual := b,
             Message := 'Values differ');

TEST_FINISHED();
END_METHOD

METHOD PRIVATE Test_ANY_LWORD_Differ
VAR
    a : LWORD := 16#0123656789ABCBEC;
    b : LWORD := 16#0123256789ABCAEE;
END_VAR
TEST('Test_ANY_LWORD_Differ');

AssertEquals(Expected := a,
             Actual := b,
             Message := 'Values differ');

TEST_FINISHED();
END_METHOD

METHOD PRIVATE Test_ANY_LWORD_Equals
VAR
    a : LWORD := 16#0123456789ABCDEF;
    b : LWORD := 16#0123456789ABCDEF;
END_VAR
TEST('Test_ANY_LWORD_Equals');

AssertEquals(Expected := a,
             Actual := b,
             Message := 'Values differ');

TEST_FINISHED();
END_METHOD

METHOD PRIVATE Test_ANY_REAL_Differ
VAR
    a : REAL := 1234.5;
    b : REAL := 1234.4;
END_VAR
TEST('Test_ANY_REAL_Differ');

AssertEquals(Expected := a,
             Actual := b,
             Message := 'Values differ');

TEST_FINISHED();
END_METHOD

METHOD PRIVATE Test_ANY_REAL_Equals
VAR
    a : REAL := 1234.5;
    b : REAL := 1234.5;
END_VAR
TEST('Test_ANY_REAL_Equals');

AssertEquals(Expected := a,
             Actual := b,
             Message := 'Values differ');

TEST_FINISHED();
END_METHOD

METHOD PRIVATE Test_ANY_SINT_Differ
VAR
    a : SINT := 127;
    b : SINT := -30;
END_VAR
TEST('Test_ANY_SINT_Differ');

AssertEquals(Expected := a,
             Actual := b,
             Message := 'Values differ');

TEST_FINISHED();
END_METHOD

METHOD PRIVATE Test_ANY_SINT_Equals
VAR
    a : SINT := -128;
    b : SINT := -128;
END_VAR
TEST('Test_ANY_SINT_Equals');

AssertEquals(Expected := a,
             Actual := b,
             Message := 'Values differ');

TEST_FINISHED();
END_METHOD

METHOD PRIVATE Test_ANY_STRING_Differ
VAR
    a : STRING := 'This is a string';
    b : STRING := 'This is another string';
END_VAR
TEST('Test_ANY_STRING_Differ');

AssertEquals(Expected := a,
             Actual := b,
             Message := 'Values differ');

TEST_FINISHED();
END_METHOD

METHOD PRIVATE Test_ANY_STRING_Equals
VAR
    a : STRING := 'Hello there';
    b : STRING := 'Hello there';
END_VAR
TEST('Test_ANY_STRING_Equals');

AssertEquals(Expected := a,
             Actual := b,
             Message := 'Values differ');

TEST_FINISHED();
END_METHOD

METHOD PRIVATE Test_ANY_TIME_Differ
VAR
    a : TIME := T#12H34M15S10MS;
    b : TIME := T#11H34M13S244MS;
END_VAR
TEST('Test_ANY_TIME_Differ');

AssertEquals(Expected := a,
             Actual := b,
             Message := 'Values differ');

TEST_FINISHED();
END_METHOD

METHOD PRIVATE Test_ANY_TIME_Equals
VAR
    a : TIME := T#11H34M13S244MS;
    b : TIME := T#11H34M13S244MS;
END_VAR
TEST('Test_ANY_TIME_Equals');

AssertEquals(Expected := a,
             Actual := b,
             Message := 'Values differ');

TEST_FINISHED();
END_METHOD

METHOD PRIVATE Test_ANY_TIME_OF_DAY_Differ
VAR
    a : TIME_OF_DAY := TIME_OF_DAY#15:36:30.123;
    b : TIME_OF_DAY := TIME_OF_DAY#06:21:11.492;
END_VAR
TEST('Test_ANY_TIME_OF_DAY_Differ');

AssertEquals(Expected := a,
             Actual := b,
             Message := 'Values differ');

TEST_FINISHED();
END_METHOD

METHOD PRIVATE Test_ANY_TIME_OF_DAY_Equals
VAR
    a : TIME_OF_DAY := TIME_OF_DAY#06:21:11.492;
    b : TIME_OF_DAY := TIME_OF_DAY#06:21:11.492;
END_VAR
TEST('Test_ANY_TIME_OF_DAY_Equals');

AssertEquals(Expected := a,
             Actual := b,
             Message := 'Values differ');

TEST_FINISHED();
END_METHOD

METHOD PRIVATE Test_ANY_UDINT_Differ
VAR
    a : UDINT := 34124214;
    b : UDINT := 52343244;
END_VAR
TEST('Test_ANY_UDINT_Differ');

AssertEquals(Expected := a,
             Actual := b,
             Message := 'Values differ');

TEST_FINISHED();
END_METHOD

METHOD PRIVATE Test_ANY_UDINT_Equals
VAR
    a : UDINT := 21845123;
    b : UDINT := 21845123;
END_VAR
TEST('Test_ANY_UDINT_Equals');

AssertEquals(Expected := a,
             Actual := b,
             Message := 'Values differ');

TEST_FINISHED();
END_METHOD

METHOD PRIVATE Test_ANY_UINT_Differ
VAR
    a : UINT := 64322;
    b : UINT := 32312;
END_VAR
TEST('Test_ANY_UINT_Differ');

AssertEquals(Expected := a,
             Actual := b,
             Message := 'Values differ');

TEST_FINISHED();
END_METHOD

METHOD PRIVATE Test_ANY_UINT_Equals
VAR
    a : UINT := 65535;
    b : UINT := 65535;
END_VAR
TEST('Test_ANY_UINT_Equals');

AssertEquals(Expected := a,
             Actual := b,
             Message := 'Values differ');

TEST_FINISHED();
END_METHOD

METHOD PRIVATE Test_ANY_ULINT_Differ
VAR
    a : ULINT := 10000;
    b : ULINT := 53685437234;
END_VAR
TEST('Test_ANY_ULINT_Differ');

AssertEquals(Expected := a,
             Actual := b,
             Message := 'Values differ');

TEST_FINISHED();
END_METHOD

METHOD PRIVATE Test_ANY_ULINT_Equals
VAR
    a : ULINT := 45683838383;
    b : ULINT := 45683838383;
END_VAR
TEST('Test_ANY_ULINT_Equals');

AssertEquals(Expected := a,
             Actual := b,
             Message := 'Values differ');

TEST_FINISHED();
END_METHOD

METHOD PRIVATE Test_ANY_USINT_Differ
VAR
    a : USINT := 3;
    b : USINT := 7;
END_VAR
TEST('Test_ANY_USINT_Differ');

AssertEquals(Expected := a,
             Actual := b,
             Message := 'Values differ');

TEST_FINISHED();
END_METHOD

METHOD PRIVATE Test_ANY_USINT_Equals
VAR
    a : USINT := 5;
    b : USINT := 5;
END_VAR
TEST('Test_ANY_USINT_Equals');

AssertEquals(Expected := a,
             Actual := b,
             Message := 'Values differ');

TEST_FINISHED();
END_METHOD

METHOD PRIVATE Test_ANY_WORD_Differ
VAR
    a : WORD := 16#EF01;
    b : WORD := 16#2345;
END_VAR
TEST('Test_ANY_WORD_Differ');

AssertEquals(Expected := a,
             Actual := b,
             Message := 'Values differ');

TEST_FINISHED();
END_METHOD

METHOD PRIVATE Test_ANY_WORD_Equals
VAR
    a : WORD := 16#ABCD;
    b : WORD := 16#ABCD;
END_VAR
TEST('Test_ANY_WORD_Equals');

AssertEquals(Expected := a,
             Actual := b,
             Message := 'Values differ');

TEST_FINISHED();
END_METHOD

END_FUNCTION_BLOCK

// ---- Test/FB_AssertEveryFailedTestTwice_ArrayVersion.TcPOU
(*
    In this testsuite we are running the same testcase over two cycles, and thus calling
    every assert method twice. This is in order to verify that we don't print every FAILED assert twice.
    With this version we are doing it with arrays.
*)
{attribute 'call_after_init'}
FUNCTION_BLOCK FB_AssertEveryFailedTestTwice_ArrayVersion EXTENDS TcUnit.FB_TestSuite
VAR
    AssertCount : USINT := 0;
END_VAR

TwiceAssertCall_Arrays();

METHOD PRIVATE TwiceAssertCall_Arrays
VAR
    aBOOL : ARRAY[0..5] OF BOOL := [TRUE, TRUE, FALSE, TRUE, FALSE, TRUE];
    bBOOL : ARRAY[0..5] OF BOOL := [TRUE, TRUE, TRUE, TRUE, FALSE, FALSE];

    aBYTE : ARRAY[0..3] OF BYTE := [16#AB, 16#AA, 16#BB, 16#89];
    bBYTE : ARRAY[0..3] OF BYTE := [16#AB, 16#CD, 16#BB, 16#89];

    aDINT : ARRAY[3..5] OF DINT := [-4746, -2147483645, 0];
    bDINT : ARRAY[3..5] OF DINT := [-4746, -2147483641, 0];

    aDWORD : ARRAY[-2..1] OF DWORD := [16#6789ABCD, 16#EFAA2346, 16#ABABABAB, 16#EEEEEEEE];
    bDWORD : ARRAY[-2..1] OF DWORD := [16#6789ABCD, 16#EF012345, 16#ABABABAB, 16#EEEEEEEE];

    aINT : ARRAY[-8..-6] OF INT := [42, -23, -32768];
    bINT : ARRAY[1..3] OF INT := [42, 24, -32768];

    aLINT : ARRAY[-1..1] OF LINT := [9_223_372_036_854_775_807, -9_223_372_036_853_775_808, 55];
    bLINT : ARRAY[4..6] OF LINT := [9_223_372_036_854_775_807, -9_223_372_036_854_775_808, 55];

    aLWORD : ARRAY[1..1] OF LWORD := [16#EDCBA09876543210];
    bLWORD : ARRAY[1..1] OF LWORD := [16#01234567890ABCDE];

    aSINT : ARRAY[0..0] OF SINT := [-128];
    bSINT : ARRAY[0..0] OF SINT := [127];

    aUDINT : ARRAY[-5..-4] OF UDINT := [4294967295, 5];
    bUDINT : ARRAY[0..1] OF UDINT := [4294967295, 4];

    aUINT : ARRAY[0..3] OF UINT := [0, 4, 8, 99];
    bUINT : ARRAY[0..3] OF UINT := [0, 4, 8, 12];

    aULINT : ARRAY[0..1] OF ULINT := [3_213_000_444_000, 9_400_000_000_000];
    bULINT : ARRAY[0..1] OF ULINT := [3_213_000_444_000, 18_446_744_073_709_551_615];

    aUSINT : ARRAY[0..10] OF USINT := [0,1,2,3,6(4),5];
    bUSINT : ARRAY[0..10] OF USINT := [0,1,2,3,6(5),6];

    aWORD : ARRAY[1..7] OF WORD := [16#2323, 16#876A, 16#4CD4, 16#F3DC, 16#BBBB, 16#FFFF, 16#1133];
    bWORD : ARRAY[1..7] OF WORD := [16#2323, 16#876A, 16#4CD4, 16#F3DC, 16#BBBB, 16#FFFF, 16#1122];
END_VAR
TEST('TwiceAssertCall_Arrays');

AssertArrayEquals_BOOL(Expecteds := aBOOL,
                       Actuals := bBOOL,
                       Message := 'Not equal BOOL');

AssertArrayEquals_BYTE(Expecteds := aBYTE,
                       Actuals := bBYTE,
                       Message := 'Not equal BYTE');

AssertArrayEquals_DINT(Expecteds := aDINT,
                       Actuals := bDINT,
                       Message := 'Not equal DINT');

AssertArrayEquals_DWORD(Expecteds := aDWORD,
                        Actuals := bDWORD,
                        Message := 'Not equal DWORD');

AssertArrayEquals_INT(Expecteds := aINT,
                      Actuals := bINT,
                      Message := 'Not equal INT');

AssertArrayEquals_LINT(Expecteds := aLINT,
                       Actuals := bLINT,
                       Message := 'Not equal LINT');

AssertArrayEquals_LWORD(Expecteds := aLWORD,
                        Actuals := bLWORD,
                        Message := 'Not equal LWORD');

AssertArrayEquals_SINT(Expecteds := aSINT,
                       Actuals := bSINT,
                       Message := 'Not equal SINT');

AssertArrayEquals_UDINT(Expecteds := aUDINT,
                        Actuals := bUDINT,
                        Message := 'Not equal UDINT');

AssertArrayEquals_UINT(Expecteds := aUINT,
                       Actuals := bUINT,
                       Message := 'Not equal UINT');

AssertArrayEquals_ULINT(Expecteds := aULINT,
                        Actuals := bULINT,
                        Message := 'Not equal ULINT');

AssertArrayEquals_USINT(Expecteds := aUSINT,
                        Actuals := bUSINT,
                        Message := 'Not equal USINT');

AssertArrayEquals_WORD(Expecteds := aWORD,
                       Actuals := bWORD,
                       Message := 'Not equal WORD');

AssertCount := AssertCount + 1;
IF AssertCount = 2 THEN
    TEST_FINISHED();
END_IF
END_METHOD

END_FUNCTION_BLOCK

// ---- Test/FB_AnyToUnionValue_Test.TcPOU
(*
    Tests the free function F_AnyToUnionValue.
*)
{attribute 'call_after_init'}
FUNCTION_BLOCK FB_AnyToUnionValue_Test EXTENDS TcUnit.FB_TestSuite IMPLEMENTS TcUnit.I_RunnableTestSuite
VAR
    Assert : TcUnit.FB_Assert;
    
    aBit : BIT := 1; // Only structures and function blocks can have BIT defined
END_VAR

METHOD FB_init : BOOL
VAR_INPUT
	bInitRetains : BOOL; // if TRUE, the retain variables are initialized (warm start / cold start)
	bInCopyCode : BOOL;  // if TRUE, the instance afterwards gets moved into the copy code (online change)
END_VAR
SUPER^.RegisterTestSuite(THIS^);
END_METHOD

METHOD RunTests : TCUNIT.E_TestSuiteRunState
Test_BOOL();
Test_BIT();
Test_BYTE();
Test_WORD();
Test_DWORD();
Test_LWORD();
Test_SINT();
Test_INT();
Test_DINT();
Test_LINT();
Test_USINT();
Test_UINT();
Test_UDINT();
Test_ULINT();
Test_REAL();
Test_LREAL();
Test_STRING();
Test_STRING_2();
Test_WSTRING();
Test_TIME();
Test_DATE();
Test_DATE_AND_TIME();
Test_TIME_OF_DAY();
Test_LTIME();

RunTests := TCUNIT.E_TestSuiteRunState.FINISHED;
END_METHOD

METHOD PRIVATE Test_BIT
VAR
    result : U_ExpectedOrActual;
END_VAR
TEST('Test_BIT');

result := TcUnit.F_AnyToUnionValue(AnyValue := aBit);

Assert.AssertEquals(Expected := aBit,
                    Actual := result.bitExpectedOrActual,
                    Message := 'Values differ');
END_METHOD

METHOD PRIVATE Test_BOOL
VAR
    a : BOOL := TRUE;
    result : U_ExpectedOrActual;
END_VAR
TEST('Test_BOOL');

result := TcUnit.F_AnyToUnionValue(AnyValue := a);

Assert.AssertEquals(Expected := a,
                    Actual := result.boolExpectedOrActual,
                    Message := 'Values differ');
END_METHOD

METHOD PRIVATE Test_BYTE
VAR
    a : BYTE := 16#8A;
    result : U_ExpectedOrActual;
END_VAR
TEST('Test_BYTE');

result := TcUnit.F_AnyToUnionValue(AnyValue := a);

Assert.AssertEquals(Expected := a,
                    Actual := result.byteExpectedOrActual,
                    Message := 'Values differ');
END_METHOD

METHOD PRIVATE Test_DATE
VAR
    a : DATE := D#2106-02-05;
    result : U_ExpectedOrActual;
END_VAR
TEST('Test_DATE');

result := TcUnit.F_AnyToUnionValue(AnyValue := a);

Assert.AssertEquals(Expected := a,
                    Actual := result.dateExpectedOrActual,
                    Message := 'Values differ');
END_METHOD

METHOD PRIVATE Test_DATE_AND_TIME
VAR
    a : DATE_AND_TIME := DT#2106-02-06-06:28:15;
    result : U_ExpectedOrActual;
END_VAR
TEST('Test_DATE_AND_TIME');

result := TcUnit.F_AnyToUnionValue(AnyValue := a);

Assert.AssertEquals(Expected := a,
                    Actual := result.dateandtimeExpectedOrActual,
                    Message := 'Values differ');
END_METHOD

METHOD PRIVATE Test_DINT
VAR
    a : DINT := 143251;
    result : U_ExpectedOrActual;
END_VAR
TEST('Test_DINT');

result := TcUnit.F_AnyToUnionValue(AnyValue := a);

Assert.AssertEquals(Expected := a,
                    Actual := result.dintExpectedOrActual,
                    Message := 'Values differ');
END_METHOD

METHOD PRIVATE Test_DWORD
VAR
    a : DWORD := 16#3456CDEF;
    result : U_ExpectedOrActual;
END_VAR
TEST('Test_DWORD');

result := TcUnit.F_AnyToUnionValue(AnyValue := a);

Assert.AssertEquals(Expected := a,
                    Actual := result.dwordExpectedOrActual,
                    Message := 'Values differ');
END_METHOD

METHOD PRIVATE Test_INT
VAR
    a : INT := -32000;
    result : U_ExpectedOrActual;
END_VAR
TEST('Test_INT');

result := TcUnit.F_AnyToUnionValue(AnyValue := a);

Assert.AssertEquals(Expected := a,
                    Actual := result.intExpectedOrActual,
                    Message := 'Values differ');
END_METHOD

METHOD PRIVATE Test_LINT
VAR
    a : LINT := -31243145;
    result : U_ExpectedOrActual;
END_VAR
TEST('Test_LINT');

result := TcUnit.F_AnyToUnionValue(AnyValue := a);

Assert.AssertEquals(Expected := a,
                    Actual := result.lintExpectedOrActual,
                    Message := 'Values differ');
END_METHOD

METHOD PRIVATE Test_LREAL
VAR
    a : LREAL := 43123923124.745423;
    result : U_ExpectedOrActual;
END_VAR
TEST('Test_LREAL');

result := TcUnit.F_AnyToUnionValue(AnyValue := a);

Assert.AssertEquals(Expected := a,
                    Actual := result.lrealExpectedOrActual,
                    Message := 'Values differ');
END_METHOD

METHOD PRIVATE Test_LTIME
VAR
    a : LTIME := LTIME#213502D23H34M33S709MS551US615NS;
    result : U_ExpectedOrActual;
END_VAR
TEST('Test_LTIME');

result := TcUnit.F_AnyToUnionValue(AnyValue := a);

Assert.AssertEquals(Expected := a,
                    Actual := result.ltimeExpectedOrActual,
                    Message := 'Values differ');
END_METHOD

METHOD PRIVATE Test_LWORD
VAR
    a : LWORD := 16#456CDEF987654321;
    result : U_ExpectedOrActual;
END_VAR
TEST('Test_LWORD');

result := TcUnit.F_AnyToUnionValue(AnyValue := a);

Assert.AssertEquals(Expected := a,
                    Actual := result.lwordExpectedOrActual,
                    Message := 'Values differ');
END_METHOD

METHOD PRIVATE Test_REAL
VAR
    a : REAL := 431239.423;
    result : U_ExpectedOrActual;
END_VAR
TEST('Test_REAL');

result := TcUnit.F_AnyToUnionValue(AnyValue := a);

Assert.AssertEquals(Expected := a,
                    Actual := result.realExpectedOrActual,
                    Message := 'Values differ');
END_METHOD

METHOD PRIVATE Test_SINT
VAR
    a : SINT := 100;
    result : U_ExpectedOrActual;
END_VAR
TEST('Test_SINT');

result := TcUnit.F_AnyToUnionValue(AnyValue := a);

Assert.AssertEquals(Expected := a,
                    Actual := result.sintExpectedOrActual,
                    Message := 'Values differ');
END_METHOD

METHOD PRIVATE Test_STRING
VAR
    a : STRING := 'This is a random string';
    result : U_ExpectedOrActual;
END_VAR
TEST('Test_STRING');

result := TcUnit.F_AnyToUnionValue(AnyValue := a);

Assert.AssertEquals(Expected := a,
                    Actual := result.stringExpectedOrActual,
                    Message := 'Values differ');
END_METHOD

METHOD PRIVATE Test_STRING_2
VAR
    a : Tc2_System.T_MaxString := '8YNn5KOmPC4dAcpOBdLWnw4WkN126EwXsj65xeurG48gWBepinNaOIKeCVMtWNBSxQWPdtUYiAusDkjMLtQhDtiWbwvmoKcFwiUGDd7pOe0fd52J7hK60oaYAX6VWWmceLJX8utaDVrVzCGXafeZLeHl6jj5enfjg4tfb2WMEBdsBuG2iDKwzwhBLCPqXDnhe5HbemIbtZT7p62OEj2oDqiIYDD6tZdlhBCCelDBx6dbIp32wFm0TpRKsTiwkZ6'; // 255 characters
    result : U_ExpectedOrActual;
END_VAR
TEST('Test_STRING_2');

result := TcUnit.F_AnyToUnionValue(AnyValue := a);

Assert.AssertEquals(Expected := a,
                    Actual := result.stringExpectedOrActual,
                    Message := 'Values differ');
END_METHOD

METHOD PRIVATE Test_TIME
VAR
    a : TIME := T#15M20S;
    result : U_ExpectedOrActual;
END_VAR
TEST('Test_TIME');

result := TcUnit.F_AnyToUnionValue(AnyValue := a);

Assert.AssertEquals(Expected := a,
                    Actual := result.timeExpectedOrActual,
                    Message := 'Values differ');
END_METHOD

METHOD PRIVATE Test_TIME_OF_DAY
VAR
    a : TIME_OF_DAY := TOD#15:36:30.123;
    result : U_ExpectedOrActual;
END_VAR
TEST('Test_TIME_OF_DAY');

result := TcUnit.F_AnyToUnionValue(AnyValue := a);

Assert.AssertEquals(Expected := a,
                    Actual := result.timeofdayExpectedOrActual,
                    Message := 'Values differ');
END_METHOD

METHOD PRIVATE Test_UDINT
VAR
    a : UDINT := 2555;
    result : U_ExpectedOrActual;
END_VAR
TEST('Test_UDINT');

result := TcUnit.F_AnyToUnionValue(AnyValue := a);

Assert.AssertEquals(Expected := a,
                    Actual := result.udintExpectedOrActual,
                    Message := 'Values differ');
END_METHOD

METHOD PRIVATE Test_UINT
VAR
    a : UINT := 34523;
    result : U_ExpectedOrActual;
END_VAR
TEST('Test_UINT');

result := TcUnit.F_AnyToUnionValue(AnyValue := a);

Assert.AssertEquals(Expected := a,
                    Actual := result.uintExpectedOrActual,
                    Message := 'Values differ');
END_METHOD

METHOD PRIVATE Test_ULINT
VAR
    a : ULINT := 25555423;
    result : U_ExpectedOrActual;
END_VAR
TEST('TEST_ULINT');

result := TcUnit.F_AnyToUnionValue(AnyValue := a);

Assert.AssertEquals(Expected := a,
                    Actual := result.ulintExpectedOrActual,
                    Message := 'Values differ');
END_METHOD

METHOD PRIVATE Test_USINT
VAR
    a : USINT := 255;
    result : U_ExpectedOrActual;
END_VAR
TEST('Test_USINT');

result := TcUnit.F_AnyToUnionValue(AnyValue := a);

Assert.AssertEquals(Expected := a,
                    Actual := result.usintExpectedOrActual,
                    Message := 'Values differ');
END_METHOD

METHOD PRIVATE Test_WORD
VAR
    a : WORD := 16#ABCD;
    result : U_ExpectedOrActual;
END_VAR
TEST('Test_WORD');

result := TcUnit.F_AnyToUnionValue(AnyValue := a);

Assert.AssertEquals(Expected := a,
                    Actual := result.wordExpectedOrActual,
                    Message := 'Values differ');
END_METHOD

METHOD PRIVATE Test_WSTRING
VAR
    a : WSTRING := "This is a random string";
    result : U_ExpectedOrActual;
END_VAR
TEST('Test_WSTRING');

result := TcUnit.F_AnyToUnionValue(AnyValue := a);

Assert.AssertEquals(Expected := a,
                    Actual := result.wstringExpectedOrActual,
                    Message := 'Values differ');
END_METHOD

END_FUNCTION_BLOCK

// ---- Test/FB_MultipleAssertWithSameParametersInSameCycleWithSameTest.TcPOU
(*
    This test-suite runs several asserts with the same parameters (same expected, actual, message) in the same cycle
    and in the same test.
    The reason we want the framework to support this is that theoretically the user could want to do an assert with the
    same message, in the same test, with the same data values for both expected and actual, although the data that the
    user does the assert on might be from different data sets.
*)
{attribute 'call_after_init'}
FUNCTION_BLOCK FB_MultipleAssertWithSameParametersInSameCycleWithSameTest EXTENDS TcUnit.FB_TestSuite

Assert_SeveralTimes();

METHOD PRIVATE Assert_SeveralTimes
VAR
    a : DWORD := 16#12345678;
    b : DWORD := 16#90ABCDEF;
    
    c : DWORD := 16#12345678;
    d : DWORD := 16#90ABCDEF;
    
    e : DWORD := 16#12345678;
    f : DWORD := 16#90ABCDEF;
END_VAR
TEST('Assert_SeveralTimes');

AssertEquals_DWORD(Expected := a,
                   Actual := b,
                   Message := 'Values differ');

AssertEquals_DWORD(Expected := c,
                   Actual := d,
                   Message := 'Values differ');

AssertEquals_DWORD(Expected := e,
                   Actual := f,
                   Message := 'Values differ');

TEST_FINISHED();
END_METHOD

END_FUNCTION_BLOCK

// ---- Test/FB_MultipleAssertWithSameParametersInDifferentCyclesButWithDifferentTests.TcPOU
(*
    This test-suite runs several asserts with the same parameters (same expected, actual, message), calling the asserts
    in different cycles and using different tests.
    On top of this, we will call new asserts (though with same parameters) in later cycles.
    The reason we want the framework to support this is that theoretically the user could want to do an assert with the
    same message, in different tests, with the same data values for both expected and actual, although the data that the
    user does the assert on might be from different data sets.
*)
{attribute 'call_after_init'}
FUNCTION_BLOCK FB_MultipleAssertWithSameParametersInDifferentCyclesButWithDifferentTests EXTENDS TcUnit.FB_TestSuite IMPLEMENTS TcUnit.I_RunnableTestSuite
VAR
    Assert : TcUnit.FB_Assert;
    TimerAgain : Tc2_Standard.TON := (PT := T#1S); // Timer to call "AssertSeveralTimesAgain"
    TimerAgainAgain : Tc2_Standard.TON := (PT := T#5S); // Timer to call "AssertSeveralTimesAgainAgain"
    CalledAll : BOOL; // Indication of whether we've called all tests
END_VAR

METHOD PRIVATE Assert_SeveralTimes
VAR
    a : DWORD := 16#12345678;
    b : DWORD := 16#90ABCDEF;

    c : DWORD := 16#12345678;
    d : DWORD := 16#90ABCDEF;

    e : DWORD := 16#12345678;
    f : DWORD := 16#90ABCDEF;
END_VAR
TEST('Assert_SeveralTimes');

Assert.AssertEquals_DWORD(Expected := a,
                          Actual := b,
                          Message := 'Values differ');

Assert.AssertEquals_DWORD(Expected := c,
                          Actual := d,
                          Message := 'Values differ');

Assert.AssertEquals_DWORD(Expected := e,
                          Actual := f,
                          Message := 'Values differ');
END_METHOD

METHOD PRIVATE Assert_SeveralTimesAgain
VAR
    a : DWORD := 16#12345678;
    b : DWORD := 16#90ABCDEF;

    c : DWORD := 16#12345678;
    d : DWORD := 16#90ABCDEF;

    e : DWORD := 16#12345678;
    f : DWORD := 16#90ABCDEF;
END_VAR
TEST('Assert_SeveralTimesAgain');

Assert.AssertEquals_DWORD(Expected := a,
                          Actual := b,
                          Message := 'Values differ');

Assert.AssertEquals_DWORD(Expected := c,
                          Actual := d,
                          Message := 'Values differ');

Assert.AssertEquals_DWORD(Expected := e,
                          Actual := f,
                          Message := 'Values differ');
END_METHOD

METHOD PRIVATE Assert_SeveralTimesAgainAgain
VAR
    a : DWORD := 16#12345678;
    b : DWORD := 16#90ABCDEF;

    c : DWORD := 16#12345678;
    d : DWORD := 16#90ABCDEF;

    e : DWORD := 16#12345678;
    f : DWORD := 16#90ABCDEF;
END_VAR
TEST('Assert_SeveralTimesAgainAgain');

Assert.AssertEquals_DWORD(Expected := a,
                          Actual := b,
                          Message := 'Values differ');

Assert.AssertEquals_DWORD(Expected := c,
                          Actual := d,
                          Message := 'Values differ');

Assert.AssertEquals_DWORD(Expected := e,
                          Actual := f,
                          Message := 'Values differ');
END_METHOD

METHOD FB_init : BOOL
VAR_INPUT
	bInitRetains : BOOL; // if TRUE, the retain variables are initialized (warm start / cold start)
	bInCopyCode : BOOL;  // if TRUE, the instance afterwards gets moved into the copy code (online change)
END_VAR
SUPER^.RegisterTestSuite(THIS^);
END_METHOD

METHOD PUBLIC RunTests : TCUNIT.E_TestSuiteRunState
TimerAgain(IN := TRUE);

Assert_SeveralTimes();

IF TimerAgain.Q THEN
    TimerAgainAgain(IN := TRUE);
    Assert_SeveralTimesAgain();
END_IF

IF TimerAgainAgain.Q THEN
    Assert_SeveralTimesAgainAgain();
    CalledAll := TRUE;
END_IF

IF CalledAll THEN
    RunTests := TCUNIT.E_TestSuiteRunState.FINISHED;
END_IF
END_METHOD

END_FUNCTION_BLOCK

// ---- Test/FB_MultipleAssertWithSameParametersInDifferentCyclesAndInSameTest.TcPOU
(*
    This test-suite runs several asserts with the same parameters (same expected, actual, message), calling the asserts
    in different cycles and using the same test.
    On top of this, we will call new asserts (though with same parameters) in later cycles.
    The reason we want the framework to support this is that theoretically the user could want to do an assert with the
    same message, using the same test with the same data values for both expected and actual, and splitting the asserts
    on different cycles.
*)
{attribute 'call_after_init'}
FUNCTION_BLOCK FB_MultipleAssertWithSameParametersInDifferentCyclesAndInSameTest EXTENDS TcUnit.FB_TestSuite IMPLEMENTS TcUnit.I_RunnableTestSuite
VAR
    Assert : TcUnit.FB_Assert;
    TimerAgain : Tc2_Standard.TON := (PT := T#1S); // Timer to call "AssertSeveralTimesAgain"
    TimerAgainAgain : Tc2_Standard.TON := (PT := T#5S); // Timer to call "AssertSeveralTimesAgainAgain"
    CalledAll : BOOL; // Indication of whether we've called all tests
END_VAR

METHOD PRIVATE Assert_SeveralTimes
VAR
    a : DWORD := 16#12345678;
    b : DWORD := 16#90ABCDEF;

    c : DWORD := 16#12345678;
    d : DWORD := 16#90ABCDEF;

    e : DWORD := 16#12345678;
    f : DWORD := 16#90ABCDEF;
    
    g : DWORD := 16#12345678;
    h : DWORD := 16#90ABCDEF;
    
    i : DWORD := 16#12345678;
    j : DWORD := 16#90ABCDEF;
    
    k : DWORD := 16#12345678;
    l : DWORD := 16#90ABCDEF;
    
    m : DWORD := 16#12345678;
    n : DWORD := 16#90ABCDEF;
    
    o : DWORD := 16#12345678;
    p : DWORD := 16#90ABCDEF;
    
    q : DWORD := 16#12345678;
    rr : DWORD := 16#90ABCDEF;
END_VAR
TEST('Assert_SeveralTimes');

Assert.AssertEquals_DWORD(Expected := a,
                          Actual := b,
                          Message := 'Values differ');
Assert.AssertEquals_DWORD(Expected := c,
                          Actual := d,
                          Message := 'Values differ');
Assert.AssertEquals_DWORD(Expected := e,
                          Actual := f,
                          Message := 'Values differ');

TimerAgain(IN := TRUE);
IF TimerAgain.Q THEN
    TimerAgainAgain(IN := TRUE);
    Assert.AssertEquals_DWORD(Expected := g,
                              Actual := h,
                              Message := 'Values differ');
    Assert.AssertEquals_DWORD(Expected := i,
                              Actual := j,
                              Message := 'Values differ');
    Assert.AssertEquals_DWORD(Expected := k,
                              Actual := l,
                              Message := 'Values differ');
END_IF

IF TimerAgainAgain.Q THEN
    Assert.AssertEquals_DWORD(Expected := m,
                              Actual := n,
                              Message := 'Values differ');
    Assert.AssertEquals_DWORD(Expected := o,
                              Actual := p,
                              Message := 'Values differ');
    Assert.AssertEquals_DWORD(Expected := q,
                              Actual := rr,
                              Message := 'Values differ');
    CalledAll := TRUE;    
END_IF
END_METHOD

METHOD FB_init : BOOL
VAR_INPUT
	bInitRetains : BOOL; // if TRUE, the retain variables are initialized (warm start / cold start)
	bInCopyCode : BOOL;  // if TRUE, the instance afterwards gets moved into the copy code (online change)
END_VAR
SUPER^.RegisterTestSuite(THIS^);
END_METHOD

METHOD PUBLIC RunTests : TCUNIT.E_TestSuiteRunState
Assert_SeveralTimes();

IF CalledAll THEN
    RunTests := TCUNIT.E_TestSuiteRunState.FINISHED;
END_IF
END_METHOD

END_FUNCTION_BLOCK
